(* Schneider Machine Expert - Basic project pump_basic_TM221CE24T, file version 3.0.0.0 *)
(* ProjectInformations: Name=Pump Basic TM221CE24T *)

HARDWARE
  Cpu 0: TM221CE24T
  EthernetConfiguration: NetworkName=M221, IpAllocationMode=ByDhcp, IpAddress=192.168.1.10, SubnetMask=255.255.255.0
  SerialLineConfiguration: Baud=Baud19200, Parity=ParityEven, DataBits=DataBits8, StopBits=StopBits1, PhysicalMedium=PhysicalMediumRs485, TransmissionMode=TransmissionModeModbusRtu, SlaveId=1, Addressing=SlaveAddressing
  MastTask: UsePeriodScanMode=false, PeriodScan=100
  FastTask: Period=255
  CpuBehavior: StartingMode=StartAsPreviousState, AutoSaveRamOnEeprom=true, WatchdogPeriod=250

SYMBOLS  (address, symbol, comment, settings)
  %M0       PUMP_RUN  "Pump running latch"
  %I0.0     PB_START
  %I0.1     PB_STOP
  %I0.2     ESTOP
  %Q0.0     PUMP_OUT

POU Pump Basic Control
  (* SectionNumber=1 *)

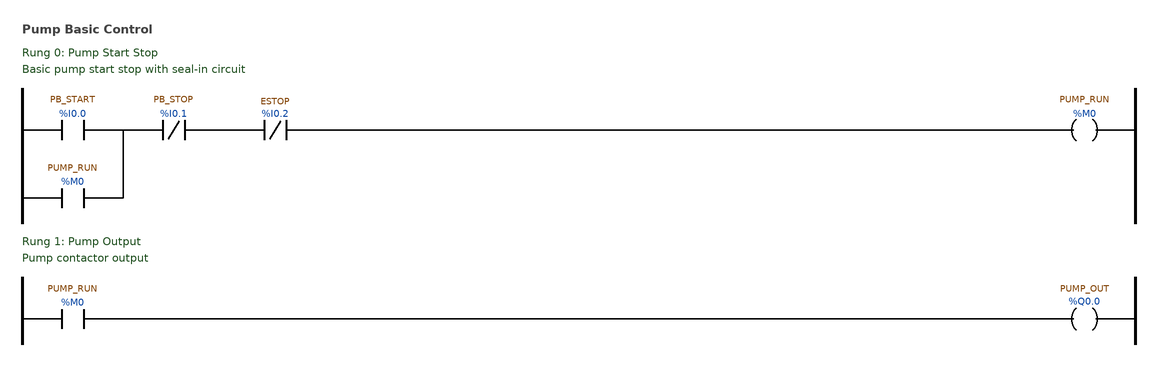

// Rung 0: Pump Start Stop
// Basic pump start stop with seal-in circuit
  LD %I0.0                (* PB_START *)
  OR %M0                  (* PUMP_RUN *)
  ANDN %I0.1              (* PB_STOP *)
  ANDN %I0.2              (* ESTOP *)
  ST %M0                  (* PUMP_RUN *)
  // as ST:
  //   PUMP_RUN := (PB_START OR PUMP_RUN) AND NOT PB_STOP AND NOT ESTOP;

// Rung 1: Pump Output
// Pump contactor output
  LD %M0                  (* PUMP_RUN *)
  ST %Q0.0                (* PUMP_OUT *)
  // as ST:
  //   PUMP_OUT := PUMP_RUN;
